PROGRAM BH0KPL_LineBackground
VAR
END_VAR

MAIN.stLine_BH0KPL.fbLine(stLine:=MAIN.stLine_BH0KPL);
MAIN.stLine_BH0KPL.stStation_BH0KPL01.fbStation(
				stLine:=MAIN.stLine_BH0KPL,
				stStation:=MAIN.stLine_BH0KPL.stStation_BH0KPL01);

END_PROGRAM

(* stored: Version 1.1.0.1, ProductVersion 3.1.4024.15
   POU BH0KPL_LineBackground: Id {03546fc4-c64b-439e-9c46-e9799456db61}, SpecialFunc None *)
